(*			
	RafalOS
	Rafał Osajda		10.11.2025		TC 4024.66
	Główny blok konfigurujący HMI
*)
FUNCTION_BLOCK FB_DefaultHMIConfiguration EXTENDS FB_Base IMPLEMENTS ITF_HMIConfiguration
VAR
END_VAR

(*			
	RafalOS
	Rafał Osajda		14.11.2025		TC 4024.66
	Dodanie do systemu menu głównego 
*)
METHOD AddMainMenu : BOOL
VAR_INPUT
	itfHMIManager	: B_HMI_Manager.ITF_HMIManagerConfigure;
END_VAR
	(*	Utowrzenie menu głównego	*)
THIS^.SetText (eLocation := E_BaseLocation.pl, wsDescription := "Okno główne");
THIS^.SetText (eLocation := E_BaseLocation.en, wsDescription := "Main screen");
THIS^.SetText (eLocation := E_BaseLocation.de, wsDescription := "Hauptbildschirm");
PRG_ControlHMI.fbMMB0_MainScreen.SetName (stName := THIS^.GetTexts ());
PRG_ControlHMI.fbMainMenu.AddButton (fbButton :=PRG_ControlHMI.fbMMB0_MainScreen);
THIS^.SetText (eLocation := E_BaseLocation.pl, wsDescription := "Receptury");
THIS^.SetText (eLocation := E_BaseLocation.en, wsDescription := "Recipe");
THIS^.SetText (eLocation := E_BaseLocation.de, wsDescription := "Rezept");
PRG_ControlHMI.fbMMB1_Recipe.SetName (stName := THIS^.GetTexts ());
PRG_ControlHMI.fbMainMenu.AddButton (fbButton :=PRG_ControlHMI.fbMMB1_Recipe);
THIS^.SetText (eLocation := E_BaseLocation.pl, wsDescription := "Parametry");
THIS^.SetText (eLocation := E_BaseLocation.en, wsDescription := "Parameters");
THIS^.SetText (eLocation := E_BaseLocation.de, wsDescription := "Parameter");
PRG_ControlHMI.fbMMB2_Parameters.SetName (stName := THIS^.GetTexts ());
PRG_ControlHMI.fbMainMenu.AddButton (fbButton :=PRG_ControlHMI.fbMMB2_Parameters);
THIS^.SetText (eLocation := E_BaseLocation.pl, wsDescription := "Zdarzenia");
THIS^.SetText (eLocation := E_BaseLocation.en, wsDescription := "Events");
THIS^.SetText (eLocation := E_BaseLocation.de, wsDescription := "Veranstaltungen");
PRG_ControlHMI.fbMMB3_Events.SetName (stName := THIS^.GetTexts ());
PRG_ControlHMI.fbMainMenu.AddButton (fbButton :=PRG_ControlHMI.fbMMB3_Events);
THIS^.SetText (eLocation := E_BaseLocation.pl, wsDescription := "Zmiana trybu");
THIS^.SetText (eLocation := E_BaseLocation.en, wsDescription := "Mode change");
THIS^.SetText (eLocation := E_BaseLocation.de, wsDescription := "Modusänderung");
PRG_ControlHMI.fbMMB4_ModeChange.SetName (stName := THIS^.GetTexts ());
PRG_ControlHMI.fbMainMenu.AddButton (fbButton :=PRG_ControlHMI.fbMMB4_ModeChange);
THIS^.SetText (eLocation := E_BaseLocation.pl, wsDescription := "Statystyki");
THIS^.SetText (eLocation := E_BaseLocation.en, wsDescription := "Statistics");
THIS^.SetText (eLocation := E_BaseLocation.de, wsDescription := "Statistiken");
PRG_ControlHMI.fbMMB5_Statistics.SetName (stName := THIS^.GetTexts ());
PRG_ControlHMI.fbMainMenu.AddButton (fbButton :=PRG_ControlHMI.fbMMB5_Statistics);
THIS^.SetText (eLocation := E_BaseLocation.pl, wsDescription := "Diagram stanów");
THIS^.SetText (eLocation := E_BaseLocation.en, wsDescription := "State diagram");
THIS^.SetText (eLocation := E_BaseLocation.de, wsDescription := "Zustandsdiagramm");
PRG_ControlHMI.fbMMB6_StateDiagram.SetName (stName := THIS^.GetTexts ());
PRG_ControlHMI.fbMainMenu.AddButton (fbButton :=PRG_ControlHMI.fbMMB6_StateDiagram);
THIS^.SetText (eLocation := E_BaseLocation.pl, wsDescription := "Ustawienia");
THIS^.SetText (eLocation := E_BaseLocation.en, wsDescription := "Settings");
THIS^.SetText (eLocation := E_BaseLocation.de, wsDescription := "Einstellungen");
PRG_ControlHMI.fbMMB7_Settings.SetName (stName := THIS^.GetTexts ());
PRG_ControlHMI.fbMainMenu.AddButton (fbButton :=PRG_ControlHMI.fbMMB7_Settings);
//
PRG_ControlHMI.fbMainMenu_HMI_Connector.AddButton (fbButtonHMI := PRG_ControlHMI.fbMMB0_MainScreen_HMI_Connector);
PRG_ControlHMI.fbMainMenu_HMI_Connector.AddButton (fbButtonHMI := PRG_ControlHMI.fbMMB1_Recipe_HMI_Connector);
PRG_ControlHMI.fbMainMenu_HMI_Connector.AddButton (fbButtonHMI := PRG_ControlHMI.fbMMB2_Parameters_HMI_Connector);
PRG_ControlHMI.fbMainMenu_HMI_Connector.AddButton (fbButtonHMI := PRG_ControlHMI.fbMMB3_Events_HMI_Connector);
PRG_ControlHMI.fbMainMenu_HMI_Connector.AddButton (fbButtonHMI := PRG_ControlHMI.fbMMB4_ModeChange_HMI_Connector);
PRG_ControlHMI.fbMainMenu_HMI_Connector.AddButton (fbButtonHMI := PRG_ControlHMI.fbMMB5_Statistics_HMI_Connector);
PRG_ControlHMI.fbMainMenu_HMI_Connector.AddButton (fbButtonHMI := PRG_ControlHMI.fbMMB6_StateDiagram_HMI_Connector);
PRG_ControlHMI.fbMainMenu_HMI_Connector.AddButton (fbButtonHMI := PRG_ControlHMI.fbMMB7_Settings_HMI_Connector);

itfHMIManager.AddMainMenuFromConfiguration (
	fbMenu := PRG_ControlHMI.fbMainMenu,
	fbMenu_HMI := PRG_ControlHMI.fbMainMenu_HMI_Connector
);
END_METHOD

(*			
	RafalOS
	Rafał Osajda		18.11.2025		TC 4024.66
	Podłączenie głównej struktury danych dla domyślnych elementów 
*)
METHOD LinkCommonStructureData : BOOL
VAR_INPUT
	itfHMIManager	: B_HMI_Manager.ITF_HMIManagerConfigure;
END_VAR
itfHMIManager.LinkHMIManagerDataFromConfiguration (stData := PRG_ControlHMI.stHMIData);
END_METHOD

METHOD LinkHMIManagerData : BOOL
VAR_INPUT
	itfHMIManager	: B_HMI_Manager.ITF_HMIManagerConfigure;
END_VAR
itfHMIManager.LinkHMIManagerDataFromConfiguration (stData := PRG_ControlHMI.stHMIData);
END_METHOD

(*			
	RafalOS
	Rafał Osajda		18.11.2025		TC 4024.66
	Ustawia przycisk na aktywny  - pierwsze okno w wyświetlaniu wizualizacji
*)
METHOD SetButtonActive : BOOL
VAR_INPUT
	itfHMIManager	: B_HMI_Manager.ITF_HMIManagerConfigure;
END_VAR
itfHMIManager.SetButtonActiveFromConfiguration (iNumber := 0, bValue := TRUE);
END_METHOD

(*			
	RafalOS
	Rafał Osajda		18.11.2025		TC 4024.66
	Ustawia przyciski na wlaczone lub wylaczone - możliwośc naciśnięcia
*)
METHOD SetButtonsEnabled : BOOL
VAR_INPUT
	itfHMIManager	: B_HMI_Manager.ITF_HMIManagerConfigure;
END_VAR

VAR
	iI					: INT;
	iNumberofButtons	: INT;
END_VAR
iNumberofButtons := itfHMIManager.GetNumberOfAddedButtons ();
FOR iI := 0 TO iNumberofButtons DO
	itfHMIManager.SetButtonsEnabledFromConfiguration (iNumber := iI, bValue := TRUE);
END_FOR
END_METHOD

(*			
	RafalOS
	Rafał Osajda		18.11.2025		TC 4024.66
	Ustawia przyciski na widoczne lub nie widoczne
*)
METHOD SetButtonsVisible : BOOL
VAR_INPUT
	itfHMIManager	: B_HMI_Manager.ITF_HMIManagerConfigure;
END_VAR
VAR
	iI					: INT;
	iNumberofButtons	: INT;
END_VAR
iNumberofButtons := itfHMIManager.GetNumberOfAddedButtons ();
FOR iI := 0 TO iNumberofButtons DO
	itfHMIManager.SetButtonsEnabledFromConfiguration (iNumber := iI, bValue := TRUE);
END_FOR
END_METHOD

END_FUNCTION_BLOCK

(* stored: Version 1.1.0.1
   POU FB_DefaultHMIConfiguration: Id {d9806d62-298f-058f-3795-91a96daea1b3}, SpecialFunc None
   Method AddMainMenu: Id {44b09da7-75f1-0fb2-248e-9ffa540d4691}
   Method LinkCommonStructureData: Id {809bebf6-2341-0229-3504-bc3941e2cafc}
   Method LinkHMIManagerData: Id {0dd4ccc1-f7b5-039f-2ef7-cc7039656273}
   Method SetButtonActive: Id {ef4dae27-eac3-0c53-0fad-accc29e40bae}
   Method SetButtonsEnabled: Id {01362e76-6df6-0e77-3a0b-ea16d9695793}
   Method SetButtonsVisible: Id {18290a14-9a2f-0158-2aba-671cc7a631d1} *)
